FUNCTION_BLOCK FB_SimulatedOutClose_DG IMPLEMENTS ITF_Regelschuif_OutClose_DG
VAR
	internalState : BOOL := FALSE;
END_VAR

{warning 'Add method implementation '}
METHOD set : BOOL
VAR_INPUT
	state : BOOL;
END_VAR
internalState := state;
END_METHOD

END_FUNCTION_BLOCK

(* stored: Version 1.1.0.1, ProductVersion 3.1.4026.8
   POU FB_SimulatedOutClose_DG: Id {ff58a706-d197-40fc-9b59-01bd0c33f601}, SpecialFunc None
   Method set: Id {e63e9833-22d7-456d-980d-87c15cf3db17} *)
